FUNCTION_BLOCK SS4_ps_Raiser_n_Flipper (* Composite FB wrapping other FBs *)
  (* Standard: 61499-2 *)
  (* Version 1.0, 2025-08-25, PS_Transformer_for_Unknown *)
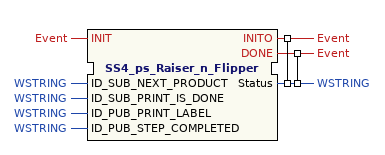
  EVENT_INPUT
    INIT; (* Initialization Request *)
  END_EVENT
  EVENT_OUTPUT
    INITO WITH Status; (* Initialization Confirm *)
    DONE WITH Status; (* Execution Confirmation *)
  END_EVENT
  VAR_INPUT
    ID_SUB_NEXT_PRODUCT : WSTRING;
    ID_SUB_PRINT_IS_DONE : WSTRING;
    ID_PUB_PRINT_LABEL : WSTRING;
    ID_PUB_STEP_COMPLETED : WSTRING;
  END_VAR
  VAR_OUTPUT
    Status : WSTRING; (* Output event qualifier *)
  END_VAR
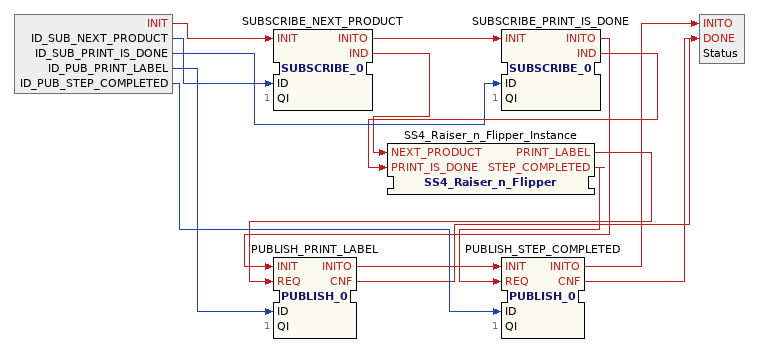
  FBS
    SS4_Raiser_n_Flipper_Instance : SS4_Raiser_n_Flipper;
    SUBSCRIBE_NEXT_PRODUCT : SUBSCRIBE_0(QI := 1);
    SUBSCRIBE_PRINT_IS_DONE : SUBSCRIBE_0(QI := 1);
    PUBLISH_PRINT_LABEL : PUBLISH_0(QI := 1);
    PUBLISH_STEP_COMPLETED : PUBLISH_0(QI := 1);
  END_FBS
  EVENT_CONNECTIONS
    INIT TO SUBSCRIBE_NEXT_PRODUCT.INIT;
    SUBSCRIBE_NEXT_PRODUCT.INITO TO SUBSCRIBE_PRINT_IS_DONE.INIT;
    SUBSCRIBE_PRINT_IS_DONE.INITO TO PUBLISH_PRINT_LABEL.INIT;
    PUBLISH_PRINT_LABEL.INITO TO PUBLISH_STEP_COMPLETED.INIT;
    PUBLISH_STEP_COMPLETED.INITO TO INITO;
    SUBSCRIBE_NEXT_PRODUCT.IND TO SS4_Raiser_n_Flipper_Instance.NEXT_PRODUCT;
    SUBSCRIBE_PRINT_IS_DONE.IND TO SS4_Raiser_n_Flipper_Instance.PRINT_IS_DONE;
    SS4_Raiser_n_Flipper_Instance.PRINT_LABEL TO PUBLISH_PRINT_LABEL.REQ;
    SS4_Raiser_n_Flipper_Instance.STEP_COMPLETED TO PUBLISH_STEP_COMPLETED.REQ;
    PUBLISH_PRINT_LABEL.CNF TO DONE;
    PUBLISH_STEP_COMPLETED.CNF TO DONE;
  END_CONNECTIONS
  DATA_CONNECTIONS
    ID_SUB_NEXT_PRODUCT TO SUBSCRIBE_NEXT_PRODUCT.ID;
    ID_SUB_PRINT_IS_DONE TO SUBSCRIBE_PRINT_IS_DONE.ID;
    ID_PUB_PRINT_LABEL TO PUBLISH_PRINT_LABEL.ID;
    ID_PUB_STEP_COMPLETED TO PUBLISH_STEP_COMPLETED.ID;
  END_CONNECTIONS
END_FUNCTION_BLOCK
